// Mitsubishi GX Works2 project: 241111_PLC_Practice1   PLC: Q02U

PROGRAM MAIN
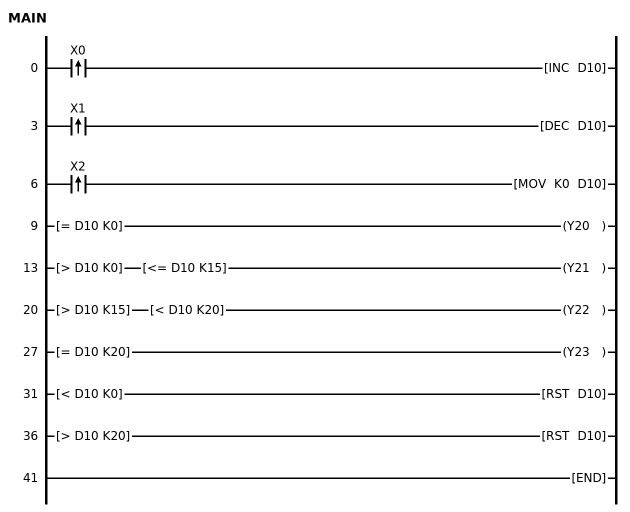
0     LDP     X0
      INC     D10
3     LDP     X1
      DEC     D10
6     LDP     X2
      MOV     K0 D10
9     LD=     D10 K0
      OUT     Y20
13    LD>     D10 K0
      AND<=   D10 K15
      OUT     Y21
20    LD>     D10 K15
      AND<    D10 K20
      OUT     Y22
27    LD=     D10 K20
      OUT     Y23
31    LD<     D10 K0
      RST     D10
36    LD>     D10 K20
      RST     D10
41    END
END_PROGRAM
